// TIA Portal V15.1 export
// export: Created 2024-05-17T05:38:29.7830472Z, ExportSetting WithDefaults, DisplayName Totally Integrated Automation Portal, DisplayVersion V15.1 Update 5, DisplayName TIA Portal Openness, DisplayVersion V15.1 Update 5, DisplayName SINAMICS Startdrive Advanced, DisplayVersion V15.1, DisplayName G130, G150, S120, S150, SINAMICS MV, S210, DisplayVersion V15.1, DisplayName G110M, G120, G120C, G120D, G120P, DisplayVersion V15.1, DisplayName STEP 7 Professional, DisplayVersion V15.1 Update 5, DisplayName STEP 7 Safety, DisplayVersion V15.1, DisplayName WinCC Professional, DisplayVersion V15.1 Update 5, DisplayName SIMATIC Visualization Architect, DisplayVersion V15.1
FUNCTION_BLOCK "LPNIODiagReadIPS7-1500"   // FB2209, SCL
TITLE = LPNIODiagReadIPS7-1500
{ S7_Optimized_Access := 'TRUE' }
AUTHOR : VCC
FAMILY : PNIODiag
VERSION : 0.0.0.0
// apette18,PADA
// stored: AutoNumber false, IsIECCheckEnabled false, IsRetainMemResEnabled false, MemoryReserve 100, SetENOAutomatically False, UDAEnableTagReadback false
   VAR_INPUT
      I_ReqIN { ExternalAccessible := 'False'; ExternalVisible := 'False'; ExternalWritable := 'False'} : Bool;
      I_HWID { ExternalAccessible := 'False'; ExternalVisible := 'False'; ExternalWritable := 'False'} : UInt := 16#64;
   END_VAR
   VAR_OUTPUT
      O_IPParam { ExternalAccessible := 'False'; ExternalVisible := 'False'; ExternalWritable := 'False'} : Struct
         IPAddress { ExternalAccessible := 'False'; ExternalVisible := 'False'; ExternalWritable := 'False'} : Array[0..3] of USInt;
         SubnetMask { ExternalAccessible := 'False'; ExternalVisible := 'False'; ExternalWritable := 'False'} : Array[0..3] of USInt;
         StandardGateway { ExternalAccessible := 'False'; ExternalVisible := 'False'; ExternalWritable := 'False'} : Array[0..3] of USInt;
         MACAddress { ExternalAccessible := 'False'; ExternalVisible := 'False'; ExternalWritable := 'False'} : Array[0..5] of USInt;
         PNName { ExternalAccessible := 'False'; ExternalVisible := 'False'; ExternalWritable := 'False'} : String;
      END_STRUCT;
      O_Busy { ExternalAccessible := 'False'; ExternalVisible := 'False'; ExternalWritable := 'False'} : Bool;
      O_Valid { ExternalAccessible := 'False'; ExternalVisible := 'False'; ExternalWritable := 'False'} : Bool;
      O_Error { ExternalAccessible := 'False'; ExternalVisible := 'False'; ExternalWritable := 'False'} : Bool;
      O_Status { ExternalAccessible := 'False'; ExternalVisible := 'False'; ExternalWritable := 'False'} : DWord;
      O_LEN { ExternalAccessible := 'False'; ExternalVisible := 'False'; ExternalWritable := 'False'} : UInt;
   END_VAR
   VAR
      ReqFlag { ExternalAccessible := 'False'; ExternalVisible := 'False'; ExternalWritable := 'False'} : Bool;
      RDREC_Status { ExternalAccessible := 'False'; ExternalVisible := 'False'; ExternalWritable := 'False'} : DWord;
      RDREC_LEN { ExternalAccessible := 'False'; ExternalVisible := 'False'; ExternalWritable := 'False'} : UInt;
      RDREC_Valid { ExternalAccessible := 'False'; ExternalVisible := 'False'; ExternalWritable := 'False'} : Bool;
      RDREC_Busy { ExternalAccessible := 'False'; ExternalVisible := 'False'; ExternalWritable := 'False'} : Bool;
      RDREC_Error { ExternalAccessible := 'False'; ExternalVisible := 'False'; ExternalWritable := 'False'} : Bool;
      StatusSave { ExternalAccessible := 'False'; ExternalVisible := 'False'; ExternalWritable := 'False'} : DWord;
      PDInterfaceDataReal { ExternalAccessible := 'False'; ExternalVisible := 'False'; ExternalWritable := 'False'} : Struct
         BlockType { ExternalAccessible := 'False'; ExternalVisible := 'False'; ExternalWritable := 'False'} : UInt;
         BlockLength { ExternalAccessible := 'False'; ExternalVisible := 'False'; ExternalWritable := 'False'} : UInt;
         BlockVersionHigh { ExternalAccessible := 'False'; ExternalVisible := 'False'; ExternalWritable := 'False'} : USInt;
         BlockVersionLow { ExternalAccessible := 'False'; ExternalVisible := 'False'; ExternalWritable := 'False'} : USInt;
         Data { ExternalAccessible := 'False'; ExternalVisible := 'False'; ExternalWritable := 'False'} : Array[0..301] of Byte;
         OwnChassisID { ExternalAccessible := 'False'; ExternalVisible := 'False'; ExternalWritable := 'False'} : String;
      END_STRUCT;
      R_TRIG { ExternalAccessible := 'False'; ExternalVisible := 'False'; ExternalWritable := 'False'; S7_SetPoint := 'True'} : R_TRIG;
      RDREC { ExternalAccessible := 'False'; ExternalVisible := 'False'; ExternalWritable := 'False'; S7_SetPoint := 'True'} : RDREC;
   END_VAR
   VAR_TEMP
      IPParValStartAddress : USInt;
      LengthOwnChassisID : USInt;
   END_VAR
BEGIN
   (*
   =================================================================================================================
   This Block is used for reading the IP Address, Subnet Mask etc. of the PLC.
   =================================================================================================================
   *)

   #R_TRIG(CLK:=#I_ReqIN,
           Q=>#ReqFlag);

   #RDREC(REQ:=#ReqFlag,
          ID:=#I_HWID,
          INDEX:=w#16#8080,
          MLEN:=300,
          VALID=>#RDREC_Valid,
          BUSY=>#RDREC_Busy,
          ERROR=>#RDREC_Error,
          STATUS=>#RDREC_Status,
          LEN=>#RDREC_LEN,
          RECORD:=#PDInterfaceDataReal);

   IF #RDREC_Valid THEN

       // Get PN-interface Name. String starts at an odd address within the array
       Chars_TO_Strg(Chars := #PDInterfaceDataReal.Data, pChars := 1, Cnt := #PDInterfaceDataReal.Data[0], Strg => #O_IPParam.PNName );

       // Calculate start address of IP-address data. Blockdata is padded to make it Unsigned32 aligned!      
       #IPParValStartAddress := #PDInterfaceDataReal.Data[0]  + (4 - ((#PDInterfaceDataReal.Data[0] + 2) MOD 4));

       // Copy MAC-Address data
       #O_IPParam.MACAddress[0] := #PDInterfaceDataReal.Data[#IPParValStartAddress + 0];
       #O_IPParam.MACAddress[1] := #PDInterfaceDataReal.Data[#IPParValStartAddress + 1];
       #O_IPParam.MACAddress[2] := #PDInterfaceDataReal.Data[#IPParValStartAddress + 2];
       #O_IPParam.MACAddress[3] := #PDInterfaceDataReal.Data[#IPParValStartAddress + 3];
       #O_IPParam.MACAddress[4] := #PDInterfaceDataReal.Data[#IPParValStartAddress + 4];
       #O_IPParam.MACAddress[5] := #PDInterfaceDataReal.Data[#IPParValStartAddress + 5];

        // Copy IP-Address data
       #O_IPParam.IPAddress[0] := #PDInterfaceDataReal.Data[#IPParValStartAddress + 8 + 0];
       #O_IPParam.IPAddress[1] := #PDInterfaceDataReal.Data[#IPParValStartAddress + 8 + 1];
       #O_IPParam.IPAddress[2] := #PDInterfaceDataReal.Data[#IPParValStartAddress + 8 + 2];
       #O_IPParam.IPAddress[3] := #PDInterfaceDataReal.Data[#IPParValStartAddress + 8 + 3];

       // Copy Subnetmask data
       #O_IPParam.SubnetMask[0] := #PDInterfaceDataReal.Data[#IPParValStartAddress + 12 + 0];
       #O_IPParam.SubnetMask[1] := #PDInterfaceDataReal.Data[#IPParValStartAddress + 12 + 1];
       #O_IPParam.SubnetMask[2] := #PDInterfaceDataReal.Data[#IPParValStartAddress + 12 + 2];
       #O_IPParam.SubnetMask[3] := #PDInterfaceDataReal.Data[#IPParValStartAddress + 12 + 3];

     // Copy Standard Gateway data
       #O_IPParam.StandardGateway[0] := #PDInterfaceDataReal.Data[#IPParValStartAddress + 16 + 0];
       #O_IPParam.StandardGateway[1] := #PDInterfaceDataReal.Data[#IPParValStartAddress + 16 + 1];
       #O_IPParam.StandardGateway[2] := #PDInterfaceDataReal.Data[#IPParValStartAddress + 16 + 2];
       #O_IPParam.StandardGateway[3] := #PDInterfaceDataReal.Data[#IPParValStartAddress + 16 + 3];

   END_IF;

   IF #RDREC_Error THEN
     // Statement section IF
     #StatusSave:=#RDREC_Status;
     #O_LEN:=0;
   ELSE
     #StatusSave:=0;
     #O_LEN:=#RDREC_LEN;
   END_IF;


   IF  #RDREC_Error OR #RDREC_Valid THEN
     // Statement section IF
     #ReqFlag:=FALSE;
   END_IF;

   #O_Status:=#StatusSave;
   #O_Valid:=#RDREC_Valid;
   #O_Busy:=#RDREC_Busy;
   #O_Error:=#RDREC_Error;
END_FUNCTION_BLOCK
